FUNCTION_BLOCK CON_LoadingStation
VAR_INPUT
	i_weighbridge : MOD_WeighBridge_Q_stOutput;
	
	i_inputbelt : MOD_InputBelt_Q_stOutput;
END_VAR
VAR_OUTPUT
	q_crane : MOD_Crane_I_stLoad;
END_VAR
VAR
END_VAR



//check if there is a truck before running. Also check for weightlimit
IF i_weighbridge.TruckOnScale AND NOT i_weighbridge.WeightLimitReached THEN
	q_crane.Ready := i_inputbelt.BoxReady;
ELSIF i_weighbridge.WeightLimitReached THEN
	q_crane.Ready := FALSE;
	//command stop
	//done loading!
ELSIF NOT i_weighbridge.TruckOnScale THEN
	q_crane.Ready := FALSE;
	//command stop //error?
	//error no truck
END_IF

END_FUNCTION_BLOCK

(* stored: Version 1.1.0.1, ProductVersion 3.1.4024.6
   POU CON_LoadingStation: Id {fd02a03d-6b4a-42d7-8b82-6be1646338cc}, SpecialFunc None *)
